// TwinCAT 3 PLC project PLC
// ProgramVersion: 3.1.4023.0
// libraries:
//   ExceptionGenerator, * (TE140x Module Vendor)
//   Tc2_Standard, * (Beckhoff Automation GmbH)
//   Tc2_System, * (Beckhoff Automation GmbH)
//   Tc2_Utilities, * (Beckhoff Automation GmbH)
//   Tc3_Module, * (Beckhoff Automation GmbH)
// project tree:
//   / PlcTask.TcTTO
//   POUs/ F_LogExecutionInfo.TcPOU, MAIN.TcPOU
// real-time tasks:
//   TASK PlcTask: cycle T#10ms, priority 20, ADS port 350

CONFIGURATION PLC
    RESOURCE PLC ON TwinCAT3
        TASK PlcTask(INTERVAL := T#10ms, PRIORITY := 20);
        PROGRAM MAIN WITH PlcTask : MAIN;
    END_RESOURCE
END_CONFIGURATION

// ---- POUs/MAIN.TcPOU
PROGRAM MAIN
VAR
	//Dynamic creation of TcCOM object
	//In this case, the required memory for the TcCOM is obtained from the router memory
	stInitfb					:ST_FB_ExceptionGenerator_TcCOM_InitStruct := (
									nOid						:= OTCID_CreateNewId,
									nTaskOid 					:= 16#02010030, //The TaskOid of the PLC task in which the wrapper is called must be specified
									nTaskSortOrder				:= 0,
									eTraceLevelMax  			:= TcTraceLevel.tlAlways,
									eModuleCaller 				:= E_MODULECALLER.Module, //The ModuleCaller must also be set to modules here
									eCallerVerification 		:= E_CallerVerification.Default,
									eStepSizeAdaptation 		:= E_StepSizeAdaptation.RequireMatchingTaskCycleTime,
									eExecutionSequence 			:= E_ExecutionSequence1.UpdateBeforeOutputMapping,
									bExecute  					:= TRUE,									
									eAccessLockState 			:= TCOM_STATE.TCOM_STATE_OP,
									eInitExceptionHandling 		:= E_FpExcptCtrlSet.ThrowExceptions,
									eUpdateExceptionHandling 	:= E_FpExcptCtrlSetEx.LogCatchAndDump
									);	
									
    
	fbExceptionGenerator 			:FB_ExceptionGenerator_TcCOM_InitStruct(stInitfb);
	stBuildInfo						:ST_ModuleBuildInfo;
	hrExecute						:HRESULT;
	
	
	//Internal data area acsess
	xReadInternalData				: BOOL;
	xWriteInternalData				: BOOL;
	stExceptionGeneratorBlockIO  	: ST_DW_ExceptionGenerator_T;
	pStExceptionGeneratorBlockIO 	: POINTER TO ST_DW_ExceptionGenerator_T;
	hr 								: HRESULT;

	//Input and outputs from the model
	Inputs							:ST_ExceptionGenerator_U_T;	//Set one of the inputs to true, to trigger an exception.
	Outputs							:ST_ExceptionGenerator_Y_T;
	                            	
	                            	
	//Execution info            	
	ExecutionInfo 					:ST_ExecutionInfo;
	PrevExecutionInfo				:ST_ExecutionInfo;
                                	
	icnt							:UDINT;
	

END_VAR

icnt:=icnt+1;

fbExceptionGenerator.bExecute; //Controls the execution of the model. 

IF 	fbExceptionGenerator.bExecute 		= TRUE 							AND
	fbExceptionGenerator.bInitialized 	= TRUE 							AND 
	fbExceptionGenerator.eObjectState 	= TCOM_STATE.TCOM_STATE_OP 
	
THEN

    // call the module
	fbExceptionGenerator(stExceptionGenerator_U:=Inputs , stExceptionGenerator_Y=>Outputs , stExecutionInfo=>ExecutionInfo );
    
	
    // handle exceptions
    IF ExecutionInfo.stActException.nExceptionCode <> 0 THEN
       // collect exception information
	   PrevExecutionInfo:=ExecutionInfo;
	   
	   //Write log message
	   stBuildInfo:=fbExceptionGenerator.stModuleBuildInfo;
	   F_LogExecutionInfo(ExecutionInfo:=ExecutionInfo,ModuleBuildInfo:=stBuildInfo);
	   
	   //Reset input data to the model - optional, but maybe a good idea to clear out any data that might have triggered the exception. 
	   //Using the TwinCAT analytics logger to cyclically log data over longer periods of time ,could be helpful in tracing the source conditions that lead to a problem..
	   //See additinal example bellow for acsessing internal data of the model.
        MEMSET(ADR(Inputs),0,SIZEOF(Inputs));
		
       // reinit TcCOM
	   //Calling the Reinit method, doesnt reset internal variables to there intial values
       fbExceptionGenerator.Reinit(stReInit :=stInitfb ); 
    END_IF
    
 END_IF
 
 
{region "ADI Interface - for acsessing internal variables"} 
	//Use with care. This shows how to acsess the internal variables ("DW" data area) of the model.
	//https://infosys.beckhoff.com/content/1033/te1400_tc3_target_matlab/11335783307.html?id=3832417987195186788
	//Might be helpful, if you for example want to re-initialize all internal variables to a know good state.
	
	// ipADI.GetImagePtr(size := , offs := adi_x := , ppData := )
	// Validate the area number "adi_x" , and offset "offs" by adding an instance of the model under TcCOM objects -> "ExceptionGenerator" -> Data Area -> "ExceptionGenerator_DW"
	
	//Read data via ADI Interface
	IF xReadInternalData THEN
		xReadInternalData:=FALSE;
		
		//Get a pointer to the data area
		hr := fbExceptionGenerator.ipADI.GetImagePtr(size := SIZEOF(stExceptionGeneratorBlockIO), offs := 0, adi_x := 2, ppData := ADR(pStExceptionGeneratorBlockIO));
		IF hr = 0 THEN
		   // copy "DW" data area to a local variable
		   MEMCPY(destAddr:=ADR(stExceptionGeneratorBlockIO),srcAddr:=pStExceptionGeneratorBlockIO,n:=SIZEOF(stExceptionGeneratorBlockIO));
		   // always release the pointer!
		   fbExceptionGenerator.ipADI.ReleaseImagePtr(pData := pStExceptionGeneratorBlockIO);
		END_IF;
			
	END_IF
	
	
	//Write data via ADI Interface
	IF xWriteInternalData THEN
		xWriteInternalData:=FALSE;
		
		//Get a pointer to the data area
		hr := fbExceptionGenerator.ipADI.GetImagePtr(size := SIZEOF(stExceptionGeneratorBlockIO), offs := 0, adi_x := 2, ppData := ADR(pStExceptionGeneratorBlockIO));
		IF hr = 0 THEN
		   //Write local data to dara area "DW" of model
		   MEMCPY(destAddr:=pStExceptionGeneratorBlockIO,srcAddr:=ADR(stExceptionGeneratorBlockIO),n:=SIZEOF(stExceptionGeneratorBlockIO));
		   // always release the pointer!
		   fbExceptionGenerator.ipADI.ReleaseImagePtr(pData := pStExceptionGeneratorBlockIO);
		END_IF;	
	END_IF
{endregion}

END_PROGRAM

// ---- POUs/F_LogExecutionInfo.TcPOU
//https://infosys.beckhoff.com/content/1033/te1400_tc3_target_matlab/11335410315.html?id=3885529162355206359
FUNCTION F_LogExecutionInfo : HRESULT
VAR_INPUT
	ExecutionInfo 				:ST_ExecutionInfo;
	ModuleBuildInfo 			:ST_ModuleBuildInfo;	
END_VAR
VAR	
	sFormatString				:STRING(255);
	sOutputString				:STRING(255);
	fbFormat					:FB_FormatString2;
 	sOut       					:T_MaxString;	
    bError     					:BOOL;
    nErrID     					:UDINT;	
	icnt						:UDINT;
	
	sExceptionCode				:T_MaxString;
	sTmxName					:T_MaxString;
	sTmxVersion					:T_MaxString;
	sReturnAddr					:T_MaxString;	
	sDumpCreated				:T_MaxString;	
	sBuildInfoTcVersion			:T_MaxString;
	sBuildInfoDebug				:T_MaxString;
	
END_VAR

//Exception code
CASE ExecutionInfo.stActException.nExceptionCode OF
	16#C000008E:
		sExceptionCode:='Divide by zero';
	16#C000008F:
		sExceptionCode:='Inexact result';
	16#C0000090:
		sExceptionCode:='Invalid operation';
	ELSE
		sExceptionCode:= TO_STRING(ExecutionInfo.stActException.nExceptionCode);
END_CASE

//Needed a string with lenght of T_MaxString
sTmxName:=ExecutionInfo.stActException.sTmxName;

//Tmx Version
sTmxVersion :=CONCAT(TO_STRING(ExecutionInfo.stActException.nTmxVersion[0]),'.');
sTmxVersion :=CONCAT(sTmxVersion,TO_STRING(ExecutionInfo.stActException.nTmxVersion[1]));
sTmxVersion	:=CONCAT(sTmxVersion,'.');
sTmxVersion :=CONCAT(sTmxVersion,TO_STRING(ExecutionInfo.stActException.nTmxVersion[2]));
sTmxVersion	:=CONCAT(sTmxVersion,'.');
sTmxVersion :=CONCAT(sTmxVersion,TO_STRING(ExecutionInfo.stActException.nTmxVersion[3]));


//Return address
sReturnAddr		:=DATA_TO_HEXSTR(ADR(ExecutionInfo.stActException.nReturnAddr),SIZEOF(ExecutionInfo.stActException.nReturnAddr),FALSE);

//Build info
sBuildInfoTcVersion		:=CONCAT(TO_STRING(ModuleBuildInfo.nTcBuild),'.');
sBuildInfoTcVersion		:=CONCAT(sBuildInfoTcVersion,TO_STRING(ModuleBuildInfo.nTcRevision));
	
IF ModuleBuildInfo.bDebug THEN
	sBuildInfoDebug:='Debug';
ELSE
	sBuildInfoDebug:='Release';
END_IF

IF ExecutionInfo.stActException.bDumpCreated THEN
	sDumpCreated:='TRUE';
ELSE
	sDumpCreated:='FALSE';
END_IF

sFormatString:=	'Exception:%s | %s:%s | Instruction Addr:0x%X | Return Addr:%s | Dump Created:%s | Cycle Count:%d | Exception Count:%d | Build info: %s %s';			 
				 
		fbFormat(
			pFormatString:=ADR(sFormatString) , 
			arg1 := F_STRING( sExceptionCode), 									//Code of the exception.
			arg2 := F_STRING( sTmxName ), 										//Name of the tmx driver that threw the exception.                                    
			arg3 := F_STRING( sTmxVersion),        								//Version of the tmx driver that threw the exception.
			arg4 := F_UDINT	( ExecutionInfo.stActException.nInstructionAddr),	//Relative address in memory; location where the exception occurred.
			arg5 := F_STRING( sReturnAddr),     								//Return addresses
			arg6 := F_STRING( sDumpCreated),		  							//TRUE if a dump file was created for the exception.
			arg7 := F_ULINT	( ExecutionInfo.nCycleCount ),  					//Current cycle count (independent of an exception)         
			arg8 := F_ULINT	( ExecutionInfo.nExceptionCount ),					//Number of exceptions that have occurred so far  
		    arg9 := F_STRING( sBuildInfoTcVersion ),						//Tc Build info Tc version
			arg10 := F_STRING( sBuildInfoDebug ),		    				// Debug or release
			pDstString:=ADR(sOutputString) , 
			nDstSize:=SIZEOF(sOutputString) , 
			bError=>bError , 
			nErrId=>nErrID );
			
	  IF NOT bError THEN
		F_LogExecutionInfo:=ADSLOGSTR( msgCtrlMask := ADSLOG_MSGTYPE_ERROR OR ADSLOG_MSGTYPE_LOG, msgFmtStr := sOutputString, strArg := '');		  
	  ELSE
		F_LogExecutionInfo:=ADSLOGSTR( msgCtrlMask := ADSLOG_MSGTYPE_ERROR OR ADSLOG_MSGTYPE_LOG, msgFmtStr := 'Error %s formating string', strArg :=TO_STRING(nErrID) );
	  END_IF
			

(*
With the InstructionAddr it is possible to judge if the exception with the given ExceptionCode always occurs at the same place in the source code. 
If the InstructionAddr is the same for repeating exceptions, it always occurs at the same point in the code. 
Via ReturnAddr you can see where the calls came from that led to the location of the exception. So you can judge if the call that leads to the exception always takes the same call path. 
If the code is called from outside the Tmx driver, there is a 0 in ReturnAddr.

*)

END_FUNCTION
